// Provides extended logger with log levels
INTERFACE I_LoggerEx EXTENDS I_Logger

// Logs the message by adding the error header to the start.
METHOD LogError
VAR_INPUT
	message	: Tc2_System.T_MaxString;
END_VAR
END_METHOD

// Logs the message by adding the info header to the start.
METHOD LogInfo
VAR_INPUT
	message	: Tc2_System.T_MaxString;
END_VAR
END_METHOD

// Gets or sets the headers which are applied to logs for their coresponding log levels.
PROPERTY LogLevelHeaders : REFERENCE TO ST_LogLevelHeaders
GET
END_GET
SET
END_SET
END_PROPERTY

// Logs the message by adding the info header to the start.
METHOD LogWarning
VAR_INPUT
	message	: Tc2_System.T_MaxString;
END_VAR
END_METHOD

END_INTERFACE

(* stored: Version 1.1.0.1, ProductVersion 3.1.4024.13
   Itf I_LoggerEx: Id {48d93d73-46a3-0e0b-1618-a89180a9d2c2}
   Method LogError: Id {2cf7cb30-c1cb-0d5f-128f-ea18bc5ed76b}
   Method LogInfo: Id {1af56a65-d4ee-0683-346e-dd528b8b4048}
   Property LogLevelHeaders: Id {f0ceafa0-0ae6-0ef7-3976-1ac588dfc336}
   Get Get: Id {f0d507bc-4cf8-07bd-38f8-ce7c11e6d8ab}
   Set Set: Id {903aa61c-91d7-05c3-0b7a-8988192f8b53}
   Method LogWarning: Id {3c88e12d-991b-0b9f-38c1-fa148bfa8609} *)
